// TIA Portal V20 export
TYPE "LKinCtrl_typePathData_advanced"
   STRUCT
      pathDataName : String["LKINCTRL_LENGTH_OF_PATHDATA_NAME"];   // name of PathData
      pointers : "LKinCtrl_typeAdvPointers";   // pointers to add / retrieve cmds in PathData
      commands : Array[1.."LKINCTRL_NO_OF_PATHDATA_ELEMENTS_ADVANCED"] of "LKinCtrl_typePathDataElement_advanced";   // command list
   END_STRUCT;
   // commands[1].cmdParameters.transitionParameters[1] := -1.0;
   // commands[2].cmdParameters.transitionParameters[1] := -1.0;
   // commands[3].cmdParameters.transitionParameters[1] := -1.0;
   // commands[4].cmdParameters.transitionParameters[1] := -1.0;
   // commands[5].cmdParameters.transitionParameters[1] := -1.0;
   // commands[6].cmdParameters.transitionParameters[1] := -1.0;
   // commands[7].cmdParameters.transitionParameters[1] := -1.0;
   // commands[8].cmdParameters.transitionParameters[1] := -1.0;
   // commands[9].cmdParameters.transitionParameters[1] := -1.0;
   // commands[10].cmdParameters.transitionParameters[1] := -1.0;
   // commands[11].cmdParameters.transitionParameters[1] := -1.0;
   // commands[12].cmdParameters.transitionParameters[1] := -1.0;
   // commands[13].cmdParameters.transitionParameters[1] := -1.0;
   // commands[14].cmdParameters.transitionParameters[1] := -1.0;
   // commands[15].cmdParameters.transitionParameters[1] := -1.0;
   // commands[16].cmdParameters.transitionParameters[1] := -1.0;
   // commands[17].cmdParameters.transitionParameters[1] := -1.0;
   // commands[18].cmdParameters.transitionParameters[1] := -1.0;
   // commands[19].cmdParameters.transitionParameters[1] := -1.0;
   // commands[20].cmdParameters.transitionParameters[1] := -1.0;
   // commands[1].parameterValid[1..4] := TRUE;
   // commands[2].parameterValid[1..4] := TRUE;
   // commands[3].parameterValid[1..4] := TRUE;
   // commands[4].parameterValid[1..4] := TRUE;
   // commands[5].parameterValid[1..4] := TRUE;
   // commands[6].parameterValid[1..4] := TRUE;
   // commands[7].parameterValid[1..4] := TRUE;
   // commands[8].parameterValid[1..4] := TRUE;
   // commands[9].parameterValid[1..4] := TRUE;
   // commands[10].parameterValid[1..4] := TRUE;
   // commands[11].parameterValid[1..4] := TRUE;
   // commands[12].parameterValid[1..4] := TRUE;
   // commands[13].parameterValid[1..4] := TRUE;
   // commands[14].parameterValid[1..4] := TRUE;
   // commands[15].parameterValid[1..4] := TRUE;
   // commands[16].parameterValid[1..4] := TRUE;
   // commands[17].parameterValid[1..4] := TRUE;
   // commands[18].parameterValid[1..4] := TRUE;
   // commands[19].parameterValid[1..4] := TRUE;
   // commands[20].parameterValid[1..4] := TRUE;
END_TYPE
